# EPICS substitutions: AutonomousMinimizationApp/Db/common/autonomous_program.substitutions
file autonomous_program.template
{
    { MODE=TEST, DEST=$(DEST), MAGPV=INTLKSUMY, MAGPV2=STATMSG,
      VACPV=INTLKSUMY, VACPV2=POSITION, CAMPV=CAMERA_PWR, CAMPV2= PNEUMATIC,
      MPS=$(MPS), TIMING=$(TIMING)
    }
}
